PROGRAM MAIN
VAR
	Timer_On_Delay: TON;
	Start: BOOL;
	QTY: INT;
END_VAR

Timer_On_Delay(IN:= Start XOR Timer_On_Delay.Q,PT:=T#1S,Q=>);
IF(Timer_On_Delay.Q)
	THEN
	//QTY++;
	//QTY+=1;
	QTY:= QTY+1;
END_IF

END_PROGRAM

(* stored: Version 1.1.0.1, ProductVersion 3.1.4024.10
   POU MAIN: Id {9bb3f490-5990-4cc7-89a0-4a301e331070}, SpecialFunc None *)
